RoboDK station: Kuka Station With Tools and Home.rdk

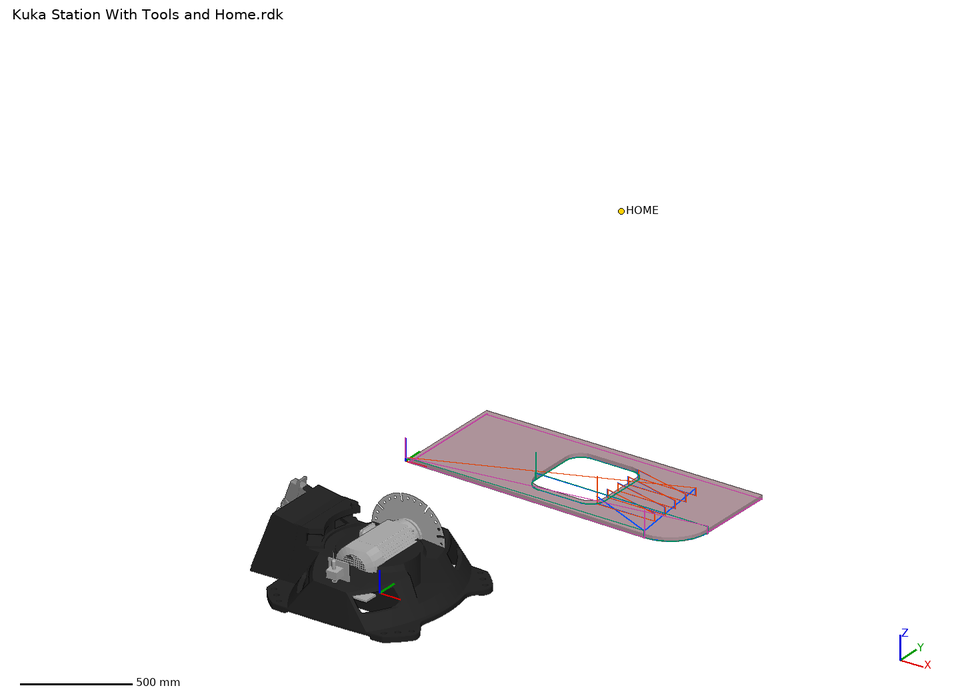
[picture v0: the station drawn from its stored meshes, robots at their saved joint values, targets as dots, program paths as lines]
Station Kuka Station With Tools and Home (saved by RoboDK 5.2.1). Poses are relative to the parent item; angles as X-Y-Z fixed-axis rotations.
  - frame KUKA KR 210 R2700 extra Base at (0, 0, 0) mm
    - robot KUKA KR 210 R2700 extra: 6 axes, payload 210 kg, reach 2696 mm, repeatability 0.06 mm, weight 1068 kg
        joint limits [-185, -140, -120, -350, -125, -350] to [185, -5, 155, 350, 125, 350]; home [0, -90, 90, 0, 0, 0]; saved at [-116.395, -62.059, 114.637, 0, 37.421, -295.134]
      - tool Circular Blade Tool, TCP at (0, 220.26, 403) mm, size 400 x 704.6 x 403 mm, geometry from Motor, Nozzle & Router Rig 2000.stl
      - tool Waterjet, TCP at (0, -363, 366) mm, rotated rx 5 ry 0 rz 0 deg
      - tool Router, TCP at (0, 325, 203) mm, rotated rx -90 ry 0 rz 0 deg
  - frame Table 1 at (-700, 1200, -20) mm
    - target HOME (Cartesian target) at (1431, -363, 1784) mm, rotated rx 0 ry 90 rz -5 deg; joints [0, -90, 90, 0, 0, 0] of KUKA KR 210 R2700 extra
  - object Top1500 US 380Vx400H 5G at (-700, 1200, -40) mm, size 1500 x 625.9 x 20 mm, geometry from Top1500 US 380Vx400H 5G.stl
  - machining project Top1500_US_380Vx400H_5G Settings: C:/Users/Curt Kilian/Dropbox/ROBOT PROGRAMMING TEST FILES/Top1500 US 380Vx400H 5G.dxf | rotZ(0) | rotX(0)*rotY(0) | rotz(0) | onStart | onPathStart | onApproach | onPoint | onRetract | onFinish | SetRPM(%1) | SetTool(%1) | Extruder(%1) | default | default | OutOnMov(%1) | OutOffMov(%1) | onPathFinish | M_RunCode(%1)
  - program Top1500_US_380Vx400H_5G (159 instructions, listed below)
  - machining project Blade Settings: C:/RoboDK/Robot Library/Top1500 US 380Vx400H 5G Blade.ngc | rotZ(0) | rotX(0)*rotY(0) | onStart | onPathStart | onApproach | onPoint | onRetract | onFinish | SetRPM(%1) | SetTool(%1) | Extruder(%1) | default | default | OutOnMov(%1) | OutOffMov(%1) | onPathFinish | M_RunCode(%1)
  - machining project Router Settings: C:/RoboDK/Robot Library/Top1500 US 380Vx400H 5G Router.ngc | rotZ(0) | rotX(0)*rotY(0) | rotz(0) | onStart | onPathStart | onApproach | onPoint | onRetract | onFinish | SetRPM(%1) | SetTool(%1) | Extruder(%1) | default | default | OutOnMov(%1) | OutOffMov(%1) | onPathFinish | M_RunCode(%1)
  - machining project Waterjet Settings: C:/RoboDK/Robot Library/Top1500 US 380Vx400H 5G Waterjet.ngc | rotZ(0) | rotX(0)*rotY(0) | rotz(0) | onStart | onPathStart | onApproach | onPoint | onRetract | onFinish | SetRPM(%1) | SetTool(%1) | Extruder(%1) | default | default | OutOnMov(%1) | OutOffMov(%1) | onPathFinish | M_RunCode(%1)
  - program Router (67 instructions, listed below)
  - program Waterjet (58 instructions, listed below)
  - program Blade (58 instructions, listed below)
  - program Prog2 (3 instructions, listed below)
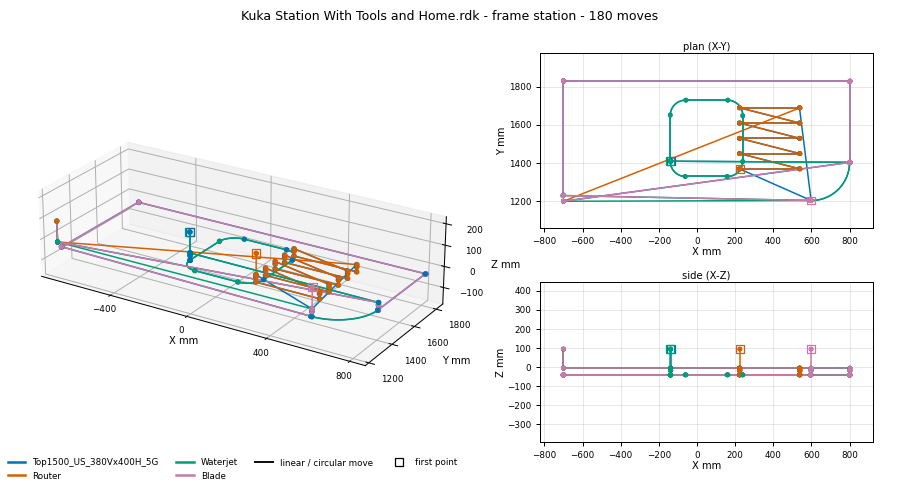
[picture p0: tool path of Kuka Station With Tools and Home.rdk in frame station, 180 of 180 moves have a stored position in this frame; points joined in program order, loops and branches not executed]

--- program Top1500_US_380Vx400H_5G (robot KUKA KR 210 R2700 extra) ---
  Smooth(1)
  Set speed (1000.0 mm/s)
  Set Ref.: Table 1
  Set Tool: Circular Blade Tool
  Show Circular Blade Tool
  MoveJ 1 to (562.5, 210, 115) mm, rotated rx 180 ry 0 rz -67.5 deg; joints [-87.471, -64.949, 119.715, 0, 35.234, 25.029]
  MoveL 2 to (562.5, 210, 115) mm, rotated rx 180 ry 0 rz -67.5 deg; joints [-87.471, -64.949, 119.715, 0, 35.234, 25.029]
  MoveL 3 to (562.5, 210, 15) mm, rotated rx 180 ry 0 rz -67.5 deg; joints [-87.471, -59.92, 119.657, 0, 30.263, 25.029]
  MoveL 4 to (562.5, 210, 15) mm, rotated rx 180 ry 0 rz -67.5 deg; joints [-87.471, -59.92, 119.657, 0, 30.263, 25.029]
  Call SetTool(1)
  Call M_RunCode(6)
  Call SetRPM(6000.0)
  Set speed (1000.0 mm/s)
  MoveL 5 to (562.5, 210, 15) mm, rotated rx 180 ry 0 rz -67.5 deg; joints [-87.471, -59.92, 119.657, 0, 30.263, 25.029]
  Call M_RunCode(3)
  MoveL 6 to (562.5, 210, 3) mm, rotated rx 180 ry 0 rz -67.5 deg; joints [-87.471, -59.3, 119.617, 0, 29.683, 25.029]
  Set speed (2.5 mm/s)
  MoveL 7 to (562.5, 210, -21) mm, rotated rx 180 ry 0 rz -90 deg; joints [-86.641, -60.19, 124.11, 0, 26.081, 3.359]
  Set speed (6.7 mm/s)
  MoveC 8 to (561.77, 211.77, -21) mm, rotated rx 180 ry 0 rz -45 deg; joints [-89.36, -56.144, 115.469, 0, 30.675, 45.64] to (560, 212.5, -21) mm, rotated rx -180 ry 0 rz 0 deg; joints [-94.901, -54.195, 111.374, 0, 32.821, 85.099]
  Set speed (2.5 mm/s)
  MoveL 9 to (560, 212.5, -20) mm, rotated rx 180 ry 0 rz 0 deg; joints [-94.901, -54.241, 111.378, 0, 32.863, 85.099]
  Set speed (6.7 mm/s)
  MoveL 10 to (560, 452.5, -20) mm, rotated rx 180 ry 0 rz -1.79 deg; joints [-94.066, -47.201, 96.831, 0, 40.37, 84.144]
  MoveC 11 to (574.27, 495.67, -20) mm, rotated rx 180 ry 0 rz -100.79 deg; joints [-86.864, -53.733, 110.317, 0, 33.416, -7.654] to (642.5, 530, -20) mm, rotated rx -180 ry 0 rz 178.21 deg; joints [-92.442, -57.698, 118.657, 0, 29.041, -94.232]
  MoveL 12 to (862.5, 530, -20) mm, rotated rx 180 ry 0 rz 178.21 deg; joints [-84.115, -57.523, 118.285, 0, 29.238, -85.905]
  MoveC 13 to (918.34, 504.8, -20) mm, rotated rx -180 ry 0 rz 133.21 deg; joints [-87.87, -56.531, 116.186, 0, 30.345, -134.66] to (940, 447.5, -20) mm, rotated rx -180 ry 0 rz 88.21 deg; joints [-89.313, -53.801, 110.459, 0, 33.342, -181.103]
  MoveL 14 to (940, 207.5, -20) mm, rotated rx -180 ry 0 rz 88.21 deg; joints [-89.196, -60.194, 124.001, 0, 26.193, -180.986]
  MoveC 15 to (914.8, 151.66, -20) mm, rotated rx -180 ry 0 rz 43.21 deg; joints [-87.577, -57.636, 118.526, 0, 29.11, -224.367] to (857.5, 130, -20) mm, rotated rx -180 ry 0 rz -1.79 deg; joints [-83.947, -56.43, 115.972, 0, 30.458, -265.737]
  MoveL 16 to (637.5, 130, -20) mm, rotated rx -180 ry 0 rz -1.79 deg; joints [-92.055, -56.636, 116.408, 0, 30.228, -273.845]
  MoveC 17 to (581.66, 155.2, -20) mm, rotated rx -180 ry 0 rz -26.79 deg; joints [-90.704, -56.615, 116.364, 0, 30.251, -297.494] to (560, 212.5, -20) mm, rotated rx 180 ry 0 rz -71.79 deg; joints [-87.324, -58.439, 120.233, 0, 28.205, -339.114]
  MoveC 18 to (561.2, 212.2, -20) mm, rotated rx -180 ry 0 rz 34.08 deg; joints [-99.338, -54.871, 112.695, 0, 32.176, -245.261] to (562.5, 210, -20) mm, rotated rx -180 ry 0 rz 50 deg; joints [-101.165, -55.817, 114.681, 0, 31.136, -231.165]
  Set speed (2.5 mm/s)
  MoveL 19 to (562.5, 210, 3) mm, rotated rx -180 ry 0 rz 90 deg; joints [-104.237, -60.41, 121.896, 0, 28.514, -194.237]
  Set speed (1000.0 mm/s)
  MoveL 20 to (562.5, 210, 15) mm, rotated rx -180 ry 0 rz 90 deg; joints [-104.237, -61.052, 121.937, 0, 29.115, -194.237]
  Call M_RunCode(9)
  MoveL 21 to (1502.5, 204.04, 15) mm, rotated rx -180 ry 0 rz 90 deg; joints [-67.477, -59.245, 118.299, 0, 30.946, -157.477]
  Call M_RunCode(3)
  MoveL 22 to (1502.5, 204.04, 3) mm, rotated rx -180 ry 0 rz 90 deg; joints [-67.477, -58.638, 118.26, 0, 30.378, -157.477]
  Set speed (2.5 mm/s)
  MoveL 23 to (1502.5, 204.04, -21) mm, rotated rx -180 ry 0 rz 90 deg; joints [-67.477, -57.415, 118.161, 0, 29.254, -157.477]
  Set speed (6.7 mm/s)
  MoveC 24 to (1501.77, 202.27, -21) mm, rotated rx -180 ry 0 rz 45 deg; joints [-67.479, -52.847, 108.561, 0, 34.286, -202.479] to (1500, 201.54, -21) mm, rotated rx -180 ry 0 rz 0 deg; joints [-63.744, -49.282, 101.181, 0, 38.1, -243.744]
  Set speed (2.5 mm/s)
  MoveL 25 to (1500, 201.54, -20) mm, rotated rx -180 ry 0 rz 0 deg; joints [-63.744, -49.323, 101.185, 0, 38.138, -243.744]
  Set speed (6.7 mm/s)
  MoveC 26 to (1438.21, 59.46, -20) mm, rotated rx 180 ry 0 rz -45.57 deg; joints [-57.647, -53.268, 109.347, 0, 33.921, -283.22] to (1293.5, 4.13, -20) mm, rotated rx 180 ry 0 rz -91.15 deg; joints [-55.853, -59.299, 122.075, 0, 27.224, -326.999]
  MoveC 27 to (1295.17, 6.46, -20) mm, rotated rx -180 ry 0 rz 34.3 deg; joints [-71.26, -58.874, 121.165, 0, 27.71, -216.958] to (1298.5, 4.08, -20) mm, rotated rx -180 ry 0 rz -19.86 deg; joints [-64.494, -56.3, 115.7, 0, 30.601, -264.351]
  Set speed (2.5 mm/s)
  MoveL 28 to (1298.5, 4.08, 3) mm, rotated rx 180 ry 0 rz 0.14 deg; joints [-67.227, -57.955, 116.863, 0, 31.092, -247.084]
  Set speed (1000.0 mm/s)
  MoveL 29 to (1298.5, 4.08, 15) mm, rotated rx -180 ry 0 rz 0.14 deg; joints [-67.227, -58.55, 116.902, 0, 31.648, -247.084]
  Call M_RunCode(9)
  MoveL 30 to (922.59, 170, 15) mm, rotated rx 180 ry 0 rz 0.14 deg; joints [-82.052, -56.815, 113.421, 0, 33.394, -261.908]
  Call M_RunCode(3)
  MoveL 31 to (922.59, 170, 3) mm, rotated rx -180 ry 0 rz 0.14 deg; joints [-82.052, -56.249, 113.384, 0, 32.866, -261.908]
  Set speed (2.5 mm/s)
  MoveL 32 to (922.59, 170, -20) mm, rotated rx -180 ry 0 rz 0.14 deg; joints [-82.052, -55.156, 113.293, 0, 31.863, -261.908]
  Set speed (6.7 mm/s)
  MoveL 33 to (1237.5, 170, -20) mm, rotated rx 180 ry 0 rz 0.14 deg; joints [-71.343, -53.125, 109.049, 0, 34.075, -251.2]
  Set speed (2.5 mm/s)
  MoveL 34 to (1237.5, 170, 3) mm, rotated rx -180 ry 0 rz 0.14 deg; joints [-71.343, -54.159, 109.137, 0, 35.022, -251.2]
  Set speed (1000.0 mm/s)
  MoveL 35 to (1237.5, 170, 15) mm, rotated rx -180 ry 0 rz 0.14 deg; joints [-71.343, -54.695, 109.173, 0, 35.522, -251.2]
  Call M_RunCode(9)
  MoveL 36 to (922.59, 250, 15) mm, rotated rx 180 ry 0 rz 0.14 deg; joints [-82.428, -54.503, 108.789, 0, 35.714, -262.285]
  Call M_RunCode(3)
  MoveL 37 to (922.59, 250, 3) mm, rotated rx 180 ry 0 rz 0.14 deg; joints [-82.428, -53.97, 108.753, 0, 35.217, -262.285]
  Set speed (2.5 mm/s)
  MoveL 38 to (922.59, 250, -20) mm, rotated rx -180 ry 0 rz 0.14 deg; joints [-82.428, -52.94, 108.666, 0, 34.274, -262.285]
  Set speed (6.7 mm/s)
  MoveL 39 to (1237.5, 250, -20) mm, rotated rx -180 ry 0 rz 0.14 deg; joints [-72.179, -50.93, 104.499, 0, 36.431, -252.035]
  Set speed (2.5 mm/s)
  MoveL 40 to (1237.5, 250, 3) mm, rotated rx -180 ry 0 rz 0.14 deg; joints [-72.179, -51.91, 104.584, 0, 37.326, -252.035]
  Set speed (1000.0 mm/s)
  MoveL 41 to (1237.5, 250, 15) mm, rotated rx -180 ry 0 rz 0.14 deg; joints [-72.179, -52.417, 104.62, 0, 37.798, -252.035]
  Call M_RunCode(9)
  MoveL 42 to (922.59, 330, 15) mm, rotated rx -180 ry 0 rz 0.14 deg; joints [-82.77, -52.117, 104.02, 0, 38.097, -262.627]
  Call M_RunCode(3)
  MoveL 43 to (922.59, 330, 3) mm, rotated rx -180 ry 0 rz 0.14 deg; joints [-82.77, -51.613, 103.985, 0, 37.629, -262.627]
  Set speed (2.5 mm/s)
  MoveL 44 to (922.59, 330, -20) mm, rotated rx 180 ry 0 rz 0.14 deg; joints [-82.77, -50.64, 103.9, 0, 36.74, -262.627]
  Set speed (6.7 mm/s)
  MoveL 45 to (1237.5, 330, -20) mm, rotated rx -180 ry 0 rz 0.14 deg; joints [-72.945, -48.643, 99.787, 0, 38.856, -252.802]
  Set speed (2.5 mm/s)
  MoveL 46 to (1237.5, 330, 3) mm, rotated rx -180 ry 0 rz 0.14 deg; joints [-72.945, -49.574, 99.87, 0, 39.703, -252.802]
  Set speed (1000.0 mm/s)
  MoveL 47 to (1237.5, 330, 15) mm, rotated rx -180 ry 0 rz 0.14 deg; joints [-72.945, -50.055, 99.905, 0, 40.15, -252.802]
  Call M_RunCode(9)
  MoveL 48 to (922.59, 410, 15) mm, rotated rx -180 ry 0 rz 0.14 deg; joints [-83.083, -49.648, 99.092, 0, 40.555, -262.94]
  Call M_RunCode(3)
  MoveL 49 to (922.59, 410, 3) mm, rotated rx -180 ry 0 rz 0.14 deg; joints [-83.083, -49.17, 99.058, 0, 40.112, -262.94]
  Set speed (2.5 mm/s)
  MoveL 50 to (922.59, 410, -20) mm, rotated rx -180 ry 0 rz 0.14 deg; joints [-83.083, -48.247, 98.975, 0, 39.272, -262.94]
  Set speed (6.7 mm/s)
  MoveL 51 to (1237.5, 410, -20) mm, rotated rx -180 ry 0 rz 0.14 deg; joints [-73.65, -46.253, 94.891, 0, 41.362, -253.506]
  Set speed (2.5 mm/s)
  MoveL 52 to (1237.5, 410, 3) mm, rotated rx 180 ry 0 rz 0.14 deg; joints [-73.65, -47.14, 94.973, 0, 42.166, -253.506]
  Set speed (1000.0 mm/s)
  MoveL 53 to (1237.5, 410, 15) mm, rotated rx -180 ry 0 rz 0.14 deg; joints [-73.65, -47.598, 95.008, 0, 42.591, -253.506]
  Call M_RunCode(9)
  MoveL 54 to (922.59, 490, 15) mm, rotated rx -180 ry 0 rz 0.14 deg; joints [-83.37, -47.082, 93.98, 0, 43.102, -263.227]
  Call M_RunCode(3)
  MoveL 55 to (922.59, 490, 3) mm, rotated rx 180 ry 0 rz 0.14 deg; joints [-83.37, -46.628, 93.946, 0, 42.682, -263.227]
  Set speed (2.5 mm/s)
  MoveL 56 to (922.59, 490, -20) mm, rotated rx -180 ry 0 rz 0.14 deg; joints [-83.37, -45.75, 93.864, 0, 41.886, -263.227]
  Set speed (6.7 mm/s)
  MoveL 57 to (1237.5, 490, -20) mm, rotated rx 180 ry 0 rz 0.14 deg; joints [-74.3, -43.747, 89.783, 0, 43.964, -254.157]
  Set speed (2.5 mm/s)
  MoveL 58 to (1237.5, 490, 3) mm, rotated rx -180 ry 0 rz 0.14 deg; joints [-74.3, -44.594, 89.865, 0, 44.729, -254.157]
  Set speed (1000.0 mm/s)
  MoveL 59 to (1237.5, 490, 15) mm, rotated rx -180 ry 0 rz 0.14 deg; joints [-74.3, -45.032, 89.899, 0, 45.133, -254.157]
  Call M_RunCode(9)
  MoveL 60 to (1298.5, 4.08, 15) mm, rotated rx 180 ry 0 rz 0.14 deg; joints [-67.227, -58.55, 116.902, 0, 31.648, -247.084]
  Call M_RunCode(3)
  MoveL 61 to (1298.5, 4.08, 3) mm, rotated rx 180 ry 0 rz 0.14 deg; joints [-67.227, -57.955, 116.863, 0, 31.092, -247.084]
  Set speed (2.5 mm/s)
  MoveL 62 to (1298.5, 4.08, -21) mm, rotated rx -180 ry 0 rz 0.14 deg; joints [-67.227, -56.757, 116.765, 0, 29.992, -247.084]
  Set speed (6.7 mm/s)
  MoveC 63 to (1296.03, 6.61, -21) mm, rotated rx -180 ry 0 rz 90.14 deg; joints [-72.695, -63.82, 132.107, 0, 21.713, -162.551] to (1293.5, 4.13, -21) mm, rotated rx -180 ry 0 rz -179.86 deg; joints [-58.877, -66.405, 138.049, 0, 18.356, -58.734]
  Set speed (2.5 mm/s)
  MoveL 64 to (1293.5, 4.13, -20) mm, rotated rx 180 ry 0 rz -179.86 deg; joints [-58.877, -66.479, 138.055, 0, 18.424, -58.734]
  Set speed (6.7 mm/s)
  MoveL 65 to (-2.5, 30.05, -20) mm, rotated rx -180 ry 0 rz -179.86 deg; joints [-124.805, -64.664, 133.87, 0, 20.794, -124.662]
  Set speed (2.5 mm/s)
  MoveL 66 to (-2.5, 30.05, -21) mm, rotated rx -180 ry 0 rz -179.86 deg; joints [-124.805, -64.597, 133.864, 0, 20.733, -124.662]
  Set speed (6.7 mm/s)
  MoveC 67 to (-1.75, 31.79, -21) mm, rotated rx -180 ry 0 rz 135.7 deg; joints [-128.538, -61.169, 126.236, 0, 24.933, -172.838] to (0, 32.5, -21) mm, rotated rx -180 ry 0 rz 91.26 deg; joints [-126.854, -57.037, 117.359, 0, 29.679, -215.593]
  Set speed (2.5 mm/s)
  MoveL 68 to (0, 32.5, -20) mm, rotated rx -180 ry 0 rz 91.26 deg; joints [-126.854, -57.088, 117.363, 0, 29.725, -215.593]
  Set speed (6.7 mm/s)
  MoveL 69 to (0, 632.5, -20) mm, rotated rx -180 ry 0 rz 91.26 deg; joints [-116.725, -41.638, 85.502, 0, 46.137, -205.464]
  Set speed (2.5 mm/s)
  MoveL 70 to (0, 632.5, -21) mm, rotated rx -180 ry 0 rz 91.26 deg; joints [-116.725, -41.603, 85.498, 0, 46.105, -205.464]
  Set speed (6.7 mm/s)
  MoveC 71 to (1.77, 631.77, -21) mm, rotated rx -180 ry 0 rz 46.26 deg; joints [-113.371, -37.427, 77.053, 0, 50.374, -247.11] to (2.5, 630, -21) mm, rotated rx -180 ry 0 rz 1.26 deg; joints [-108.91, -37.206, 76.607, 0, 50.598, -287.649]
  Set speed (2.5 mm/s)
  MoveL 72 to (2.5, 630, -20) mm, rotated rx 180 ry 0 rz 1.26 deg; joints [-108.91, -37.239, 76.612, 0, 50.628, -287.649]
  Set speed (6.7 mm/s)
  MoveL 73 to (1502.5, 630, -20) mm, rotated rx -180 ry 0 rz 1.26 deg; joints [-68.741, -35.972, 74.058, 0, 51.913, -247.48]
  Set speed (2.5 mm/s)
  MoveL 74 to (1502.5, 630, -21) mm, rotated rx -180 ry 0 rz 1.26 deg; joints [-68.741, -35.939, 74.054, 0, 51.885, -247.48]
  Set speed (6.7 mm/s)
  MoveC 75 to (1501.77, 628.23, -21) mm, rotated rx 180 ry 0 rz -43.74 deg; joints [-64.356, -35.758, 73.69, 0, 52.068, -288.095] to (1500, 627.5, -21) mm, rotated rx 180 ry 0 rz -88.74 deg; joints [-60.892, -39.799, 81.844, 0, 47.955, -329.631]
  Set speed (2.5 mm/s)
  MoveL 76 to (1500, 627.5, -20) mm, rotated rx 180 ry 0 rz -88.74 deg; joints [-60.892, -39.834, 81.849, 0, 47.985, -329.631]
  Set speed (6.7 mm/s)
  MoveL 77 to (1500, 201.54, -20) mm, rotated rx 180 ry 0 rz -88.74 deg; joints [-54.043, -51.428, 105.528, 0, 35.9, -322.782]
  MoveC 78 to (1501.77, 202.27, -20) mm, rotated rx 180 ry 0 rz -43.74 deg; joints [-58.574, -48.672, 99.847, 0, 38.825, -282.313] to (1502.5, 204.04, -20) mm, rotated rx -180 ry 0 rz 1.26 deg; joints [-63.845, -49.288, 101.113, 0, 38.175, -242.584]
  Set speed (2.5 mm/s)
  MoveL 79 to (1502.5, 204.04, 3) mm, rotated rx 180 ry 0 rz 1.26 deg; joints [-63.845, -50.232, 101.197, 0, 39.035, -242.584]
  Set speed (1000.0 mm/s)
  MoveL 80 to (1502.5, 204.04, 15) mm, rotated rx -180 ry 0 rz 1.26 deg; joints [-63.845, -50.72, 101.232, 0, 39.489, -242.584]
  Call M_RunCode(9)
  MoveL 81 to (0, 0, 15) mm, rotated rx 180 ry 0 rz 1.26 deg; joints [-116.395, -57.394, 114.582, 0, 32.812, -295.134]
  MoveL 82 to (0, 0, 15) mm, rotated rx 180 ry 0 rz 1.26 deg; joints [-116.395, -57.394, 114.582, 0, 32.812, -295.134]
  MoveL 83 to (0, 0, 115) mm, rotated rx 180 ry 0 rz 1.26 deg; joints [-116.395, -62.059, 114.637, 0, 37.421, -295.134]
  Call M_RunCode(2)

--- program Router (robot KUKA KR 210 R2700 extra) ---
  Smooth(1)
  Set speed (1000.0 mm/s)
  Set Ref.: Table 1
  Set Tool: Router
  Show Router
  MoveJ 1 to (925.09, 170, 115) mm, rotated rx -180 ry 0 rz -180 deg; joints [-82.825, -42.749, 100.39, 8.476, 122.075, -85.475]
  MoveL 2 to (925.09, 170, 115) mm, rotated rx -180 ry 0 rz -180 deg; joints [-82.825, -42.749, 100.39, 8.476, 122.075, -85.475]
  MoveL 3 to (925.09, 170, 15) mm, rotated rx -180 ry 0 rz -180 deg; joints [-82.825, -38.29, 99.098, 8.206, 118.942, -86.008]
  MoveL 4 to (925.09, 170, 15) mm, rotated rx -180 ry 0 rz -180 deg; joints [-82.825, -38.29, 99.098, 8.206, 118.942, -86.008]
  Call SetTool(10)
  Call M_RunCode(6)
  Call SetRPM(6000.0)
  Set speed (1000.0 mm/s)
  MoveL 5 to (925.09, 170, 15) mm, rotated rx -180 ry 0 rz -180 deg; joints [-82.825, -38.29, 99.098, 8.206, 118.942, -86.008]
  Call M_RunCode(3)
  MoveL 6 to (925.09, 170, 3) mm, rotated rx -180 ry 0 rz -180 deg; joints [-82.825, -37.747, 98.915, 8.178, 118.586, -86.067]
  Set speed (2.5 mm/s)
  MoveL 7 to (925.09, 170, -20) mm, rotated rx -180 ry 0 rz -180 deg; joints [-82.825, -36.704, 98.547, 8.126, 117.917, -86.175]
  MoveL 8 to (1240, 170, -20) mm, rotated rx 180 ry 0 rz 180 deg; joints [-73.195, -35.178, 94.456, 19.357, 119.278, -80.251]
  MoveL 9 to (1240, 170, 3) mm, rotated rx -180 ry 0 rz 180 deg; joints [-73.195, -36.186, 94.82, 19.479, 119.886, -80.005]
  Set speed (1000.0 mm/s)
  MoveL 10 to (1240, 170, 15) mm, rotated rx -180 ry 0 rz -14.25 deg; joints [-65.63, -47.18, 138.68, 190.12, 91.477, -89.736]
  Call M_RunCode(9)
  MoveL 11 to (925.09, 250, 15) mm, rotated rx -180 ry 0 rz -14.25 deg; joints [-83.331, -47.144, 139.017, 172.411, 91.857, -90.247]
  Call M_RunCode(3)
  MoveL 12 to (925.09, 250, 3) mm, rotated rx 180 ry 0 rz -14.25 deg; joints [-83.331, -46.199, 138.732, 172.408, 92.511, -90.335]
  Set speed (2.5 mm/s)
  MoveL 13 to (925.09, 250, -20) mm, rotated rx -180 ry 0 rz 180 deg; joints [-83.129, -34.844, 93.582, 8.024, 121.012, -85.846]
  MoveL 14 to (1240, 250, -20) mm, rotated rx 180 ry 0 rz 180 deg; joints [-73.877, -33.246, 89.489, 19.173, 122.263, -79.485]
  MoveL 15 to (1240, 250, 3) mm, rotated rx -180 ry 0 rz 180 deg; joints [-73.877, -34.217, 89.851, 19.301, 122.839, -79.247]
  Set speed (1000.0 mm/s)
  MoveL 16 to (1240, 250, 15) mm, rotated rx -180 ry 0 rz -14.25 deg; joints [-67.3, -47.34, 135.225, 188.452, 87.908, -90.311]
  Call M_RunCode(9)
  MoveL 17 to (925.09, 330, 15) mm, rotated rx 180 ry 0 rz -14.25 deg; joints [-83.802, -47.34, 135.279, 171.939, 87.959, -89.711]
  Call M_RunCode(3)
  MoveL 18 to (925.09, 330, 3) mm, rotated rx 180 ry 0 rz -14.25 deg; joints [-83.802, -46.462, 135.015, 171.942, 88.567, -89.797]
  Set speed (2.5 mm/s)
  MoveL 19 to (925.09, 330, -20) mm, rotated rx -180 ry 0 rz 180 deg; joints [-83.409, -32.809, 88.393, 7.973, 124.157, -85.503]
  MoveL 20 to (1240, 330, -20) mm, rotated rx -180 ry 0 rz -160 deg; joints [-78.333, -32.745, 88.233, 36.817, 118.831, -70.152]
  MoveL 21 to (1240, 330, 3) mm, rotated rx 180 ry 0 rz -160 deg; joints [-78.333, -33.708, 88.595, 37.018, 119.311, -69.739]
  Set speed (1000.0 mm/s)
  MoveL 22 to (1240, 330, 15) mm, rotated rx 180 ry 0 rz -14.25 deg; joints [-68.766, -47.168, 131.631, 187.013, 84.504, -90.675]
  Call M_RunCode(9)
  MoveL 23 to (925.09, 410, 15) mm, rotated rx -180 ry 0 rz -14.25 deg; joints [-84.21, -47.15, 131.423, 171.494, 84.336, -89.154]
  Call M_RunCode(3)
  MoveL 24 to (925.09, 410, 3) mm, rotated rx 180 ry 0 rz -14.25 deg; joints [-84.21, -46.33, 131.176, 171.502, 84.902, -89.239]
  Set speed (2.5 mm/s)
  MoveL 25 to (925.09, 410, -20) mm, rotated rx -180 ry 0 rz -160 deg; joints [-87.652, -31.618, 85.445, 26.989, 123.086, -74.463]
  MoveL 26 to (1240, 410, -20) mm, rotated rx 180 ry 0 rz -160 deg; joints [-78.787, -30.55, 82.849, 37.446, 121.535, -68.172]
  MoveL 27 to (1240, 410, 3) mm, rotated rx -180 ry 0 rz -160 deg; joints [-78.787, -31.48, 83.212, 37.66, 121.985, -67.765]
  Set speed (1000.0 mm/s)
  MoveL 28 to (1240, 410, 15) mm, rotated rx 180 ry 0 rz -14.25 deg; joints [-70.061, -46.714, 127.907, 185.752, 81.237, -90.879]
  Call M_RunCode(9)
  MoveL 29 to (925.09, 490, 15) mm, rotated rx 180 ry 0 rz -14.25 deg; joints [-84.569, -46.643, 127.455, 171.065, 80.922, -88.579]
  Call M_RunCode(3)
  MoveL 30 to (925.09, 490, 3) mm, rotated rx -180 ry 0 rz -14.25 deg; joints [-84.569, -45.876, 127.222, 171.078, 81.45, -88.663]
  Set speed (2.5 mm/s)
  MoveL 31 to (925.09, 490, -20) mm, rotated rx -180 ry 0 rz 140 deg; joints [-76.2, -29.713, 80.842, 327.707, 124.27, -109.589]
  MoveL 32 to (1240, 490, -20) mm, rotated rx -180 ry 0 rz 120 deg; joints [-64.593, -28.718, 78.484, 317.905, 122.122, -115.658]
  MoveL 33 to (1240, 490, 3) mm, rotated rx 180 ry 0 rz 120 deg; joints [-64.593, -29.627, 78.851, 317.675, 122.523, -116.089]
  Set speed (1000.0 mm/s)
  MoveL 34 to (1240, 490, 15) mm, rotated rx 180 ry 0 rz 21.56 deg; joints [-61.941, -44.525, 117.868, 230.829, 79.299, -102.839]
  Call M_RunCode(9)
  MoveL 35 to (0, 0, 15) mm, rotated rx -180 ry 0 rz 21.56 deg; joints [-123.96, -46.528, 142.379, 167.539, 95.714, -91.26]
  MoveL 36 to (0, 0, 15) mm, rotated rx -180 ry 0 rz 21.56 deg; joints [-123.96, -46.528, 142.379, 167.539, 95.714, -91.26]
  MoveL 37 to (0, 0, 115) mm, rotated rx 180 ry 0 rz 21.56 deg; joints [-123.96, -55.295, 144.61, 167.601, 89.332, -89.853]
  Call M_RunCode(2)

--- program Waterjet (robot KUKA KR 210 R2700 extra) ---
  Smooth(1)
  Set speed (1000.0 mm/s)
  Set Ref.: Table 1
  Set Tool: Waterjet
  Show Waterjet
  MoveJ 1 to (560.5, 210, 115) mm, rotated rx 180 ry 0 rz -180 deg; joints [-94.634, -57.138, 106.366, 0.69, 35.79, -95.176]
  MoveL 2 to (560.5, 210, 115) mm, rotated rx 180 ry 0 rz -180 deg; joints [-94.634, -57.138, 106.366, 0.69, 35.79, -95.176]
  MoveL 3 to (560.5, 210, 15) mm, rotated rx -180 ry 0 rz -180 deg; joints [-94.634, -52.933, 106.28, 0.768, 31.671, -95.271]
  MoveL 4 to (560.5, 210, 15) mm, rotated rx -180 ry 0 rz -180 deg; joints [-94.634, -52.933, 106.28, 0.768, 31.671, -95.271]
  Call SetTool(2)
  Call M_RunCode(6)
  Call SetRPM(6000.0)
  Set speed (1000.0 mm/s)
  MoveL 5 to (560.5, 210, 15) mm, rotated rx -180 ry 0 rz -180 deg; joints [-94.634, -52.933, 106.28, 0.768, 31.671, -95.271]
  Call M_RunCode(3)
  MoveL 6 to (560.5, 210, 3) mm, rotated rx -180 ry 0 rz -180 deg; joints [-94.634, -52.414, 106.241, 0.779, 31.192, -95.283]
  Set speed (2.5 mm/s)
  MoveL 7 to (560.5, 210, -21) mm, rotated rx 180 ry 0 rz -180 deg; joints [-94.634, -51.368, 106.142, 0.801, 30.244, -95.309]
  Set speed (4.2 mm/s)
  MoveC 8 to (560.35, 210.35, -21) mm, rotated rx -180 ry 0 rz 180 deg; joints [-94.638, -51.357, 106.121, 0.801, 30.255, -95.313] to (560, 210.5, -21) mm, rotated rx -180 ry 0 rz -180 deg; joints [-94.649, -51.352, 106.11, 0.803, 30.261, -95.326]
  Set speed (2.5 mm/s)
  MoveL 9 to (560, 210.5, -20) mm, rotated rx -180 ry 0 rz -180 deg; joints [-94.649, -51.396, 106.115, 0.802, 30.3, -95.324]
  Set speed (4.2 mm/s)
  MoveL 10 to (560, 450.5, -20) mm, rotated rx 180 ry 0 rz 180 deg; joints [-94.083, -44.054, 90.955, 0.576, 38.114, -94.52]
  MoveC 11 to (583.79, 506.92, -20) mm, rotated rx 180 ry 0 rz -180 deg; joints [-93.296, -42.224, 87.217, 0.447, 40.016, -93.626] to (640.5, 530, -20) mm, rotated rx 180 ry 0 rz -180 deg; joints [-91.67, -41.519, 85.779, 0.223, 40.742, -91.832]
  MoveL 12 to (860.5, 530, -20) mm, rotated rx 180 ry 0 rz 180 deg; joints [-85.504, -41.331, 85.396, -0.597, 40.951, -85.069]
  MoveC 13 to (916.92, 506.21, -20) mm, rotated rx -180 ry 0 rz -180 deg; joints [-83.862, -41.966, 86.69, -0.825, 40.307, -83.256] to (940, 449.5, -20) mm, rotated rx 180 ry 0 rz -180 deg; joints [-83.021, -43.77, 90.372, -0.976, 38.438, -82.282]
  MoveL 14 to (940, 209.5, -20) mm, rotated rx -180 ry 0 rz -180 deg; joints [-82.059, -51.108, 105.514, -1.353, 30.649, -80.924]
  MoveC 15 to (916.21, 153.08, -20) mm, rotated rx 180 ry 0 rz -180 deg; joints [-82.597, -52.794, 109.04, -1.336, 28.801, -81.454] to (859.5, 130, -20) mm, rotated rx -180 ry 0 rz -180 deg; joints [-84.448, -53.613, 110.763, -1.033, 27.877, -83.556]
  MoveL 16 to (639.5, 130, -20) mm, rotated rx -180 ry 0 rz 180 deg; joints [-92.111, -53.796, 111.149, 0.396, 27.651, -92.455]
  MoveC 17 to (583.08, 153.79, -20) mm, rotated rx 180 ry 0 rz -180 deg; joints [-94.017, -53.051, 109.581, 0.734, 28.484, -94.647] to (560, 210.5, -20) mm, rotated rx -180 ry 0 rz -180 deg; joints [-94.649, -51.396, 106.115, 0.802, 30.3, -95.324]
  MoveC 18 to (560.35, 210.35, -20) mm, rotated rx 180 ry 0 rz -180 deg; joints [-94.638, -51.401, 106.125, 0.8, 30.295, -95.312] to (560.5, 210, -20) mm, rotated rx 180 ry 0 rz -180 deg; joints [-94.634, -51.412, 106.147, 0.8, 30.283, -95.308]
  Set speed (2.5 mm/s)
  MoveL 19 to (560.5, 210, 3) mm, rotated rx -180 ry 0 rz -180 deg; joints [-94.634, -52.414, 106.241, 0.779, 31.192, -95.283]
  Set speed (1000.0 mm/s)
  MoveL 20 to (560.5, 210, 15) mm, rotated rx -180 ry 0 rz -180 deg; joints [-94.634, -52.933, 106.28, 0.768, 31.671, -95.271]
  Call M_RunCode(9)
  MoveL 21 to (1500.5, 204.04, 15) mm, rotated rx 180 ry 0 rz 180 deg; joints [-64.979, -47.787, 95.944, -3.483, 37.361, -62.293]
  Call M_RunCode(3)
  MoveL 22 to (1500.5, 204.04, 3) mm, rotated rx 180 ry 0 rz 180 deg; joints [-64.979, -47.322, 95.906, -3.517, 36.936, -62.25]
  Set speed (2.5 mm/s)
  MoveL 23 to (1500.5, 204.04, -21) mm, rotated rx 180 ry 0 rz 180 deg; joints [-64.979, -46.385, 95.812, -3.588, 36.094, -62.162]
  Set speed (4.2 mm/s)
  MoveC 24 to (1500.35, 203.69, -21) mm, rotated rx 180 ry 0 rz 180 deg; joints [-64.978, -46.397, 95.836, -3.589, 36.081, -62.16] to (1500, 203.54, -21) mm, rotated rx -180 ry 0 rz -180 deg; joints [-64.986, -46.406, 95.855, -3.589, 36.071, -62.168]
  Set speed (2.5 mm/s)
  MoveL 25 to (1500, 203.54, -20) mm, rotated rx 180 ry 0 rz -180 deg; joints [-64.986, -46.445, 95.859, -3.586, 36.106, -62.172]
  Set speed (4.2 mm/s)
  MoveC 26 to (1439.64, 60.86, -20) mm, rotated rx -180 ry 0 rz -180 deg; joints [-64.8, -51.107, 105.512, -4.116, 31.134, -61.36] to (1295.5, 4.09, -20) mm, rotated rx 180 ry 0 rz 180 deg; joints [-68.543, -54.187, 111.974, -3.944, 27.614, -65.121]
  MoveC 27 to (1296.01, 4.58, -20) mm, rotated rx 180 ry 0 rz -180 deg; joints [-68.532, -54.169, 111.937, -3.943, 27.634, -65.112] to (1296.5, 4.08, -20) mm, rotated rx 180 ry 0 rz -180 deg; joints [-68.51, -54.177, 111.954, -3.948, 27.626, -65.085]
  Set speed (2.5 mm/s)
  MoveL 28 to (1296.5, 4.08, 3) mm, rotated rx 180 ry 0 rz 180 deg; joints [-68.51, -55.255, 112.051, -3.824, 28.604, -65.226]
  Set speed (1000.0 mm/s)
  MoveL 29 to (1296.5, 4.08, 15) mm, rotated rx -180 ry 0 rz 180 deg; joints [-68.51, -55.813, 112.092, -3.762, 29.12, -65.296]
  Call M_RunCode(9)
  MoveL 30 to (0, 0, 15) mm, rotated rx -180 ry 0 rz 180 deg; joints [-114.857, -54.743, 109.93, 4.159, 30.34, -118.365]
  MoveL 31 to (0, 0, 15) mm, rotated rx -180 ry 0 rz 180 deg; joints [-114.857, -54.743, 109.93, 4.159, 30.34, -118.365]
  MoveL 32 to (0, 0, 115) mm, rotated rx -180 ry 0 rz -180 deg; joints [-114.857, -59.143, 110.017, 3.695, 34.642, -117.815]
  Call M_RunCode(2)

--- program Blade (robot KUKA KR 210 R2700 extra) ---
  Smooth(1)
  Set speed (1000.0 mm/s)
  Set Ref.: Table 1
  Set Tool: Circular Blade Tool
  Show Circular Blade Tool
  MoveJ 1 to (1298.5, 4.08, 115) mm, rotated rx 180 ry 0 rz -45.57 deg; joints [-60.906, -63.063, 116.413, 0, 36.65, 73.521]
  MoveL 2 to (1298.5, 4.08, 115) mm, rotated rx 180 ry 0 rz -45.57 deg; joints [-60.906, -63.063, 116.413, 0, 36.65, 73.521]
  MoveL 3 to (1298.5, 4.08, 15) mm, rotated rx 180 ry 0 rz -45.57 deg; joints [-60.906, -58.278, 116.356, 0, 31.922, 73.521]
  MoveL 4 to (1298.5, 4.08, 15) mm, rotated rx 180 ry 0 rz -45.57 deg; joints [-60.906, -58.278, 116.356, 0, 31.922, 73.521]
  Call SetTool(1)
  Call M_RunCode(6)
  Call SetRPM(6000.0)
  Set speed (1000.0 mm/s)
  MoveL 5 to (1298.5, 4.08, 15) mm, rotated rx 180 ry 0 rz -45.57 deg; joints [-60.906, -58.278, 116.356, 0, 31.922, 73.521]
  Call M_RunCode(3)
  MoveL 6 to (1298.5, 4.08, 3) mm, rotated rx -180 ry 0 rz -45.57 deg; joints [-60.906, -57.688, 116.318, 0, 31.371, 73.521]
  Set speed (2.5 mm/s)
  MoveL 7 to (1298.5, 4.08, -21) mm, rotated rx -180 ry 0 rz -0.57 deg; joints [-67.133, -56.729, 116.705, 0, 30.024, 112.294]
  Set speed (6.7 mm/s)
  MoveC 8 to (1296.03, 6.61, -21) mm, rotated rx -180 ry 0 rz 89.43 deg; joints [-72.731, -63.758, 131.968, 0, 21.79, 196.696] to (1293.5, 4.13, -21) mm, rotated rx -180 ry 0 rz 179.43 deg; joints [-58.995, -66.436, 138.122, 0, 18.314, 300.432]
  Set speed (2.5 mm/s)
  MoveL 9 to (1293.5, 4.13, -20) mm, rotated rx 180 ry 0 rz 178.85 deg; joints [-59.09, -66.534, 138.185, 0, 18.349, 299.764]
  Set speed (6.7 mm/s)
  MoveL 10 to (-2.5, 30.05, -20) mm, rotated rx -180 ry 0 rz 178.85 deg; joints [-124.993, -64.598, 133.719, 0, 20.879, 233.861]
  Set speed (2.5 mm/s)
  MoveL 11 to (-2.5, 30.05, -21) mm, rotated rx -180 ry 0 rz 178.86 deg; joints [-124.992, -64.531, 133.715, 0, 20.816, 233.871]
  Set speed (6.7 mm/s)
  MoveC 12 to (-1.75, 31.79, -21) mm, rotated rx -180 ry 0 rz 134.42 deg; joints [-128.561, -61.047, 125.972, 0, 25.076, 185.858] to (0, 32.5, -21) mm, rotated rx -180 ry 0 rz 89.98 deg; joints [-126.746, -56.932, 117.135, 0, 29.797, 143.235]
  Set speed (2.5 mm/s)
  MoveL 13 to (0, 32.5, -20) mm, rotated rx -180 ry 0 rz 90 deg; joints [-126.747, -56.984, 117.143, 0, 29.841, 143.253]
  Set speed (6.7 mm/s)
  MoveL 14 to (0, 632.5, -20) mm, rotated rx -180 ry 0 rz 90 deg; joints [-116.665, -41.487, 85.194, 0, 46.292, 153.335]
  Set speed (2.5 mm/s)
  MoveL 15 to (0, 632.5, -21) mm, rotated rx 180 ry 0 rz 90 deg; joints [-116.665, -41.451, 85.19, 0, 46.261, 153.335]
  Set speed (6.7 mm/s)
  MoveC 16 to (1.77, 631.77, -21) mm, rotated rx -180 ry 0 rz 45 deg; joints [-113.252, -37.357, 76.911, 0, 50.445, 111.748] to (2.5, 630, -21) mm, rotated rx 180 ry 0 rz 0 deg; joints [-108.788, -37.264, 76.724, 0, 50.54, 71.212]
  Set speed (2.5 mm/s)
  MoveL 17 to (2.5, 630, -20) mm, rotated rx 180 ry 0 rz 0 deg; joints [-108.788, -37.297, 76.728, 0, 50.569, 71.212]
  Set speed (6.7 mm/s)
  MoveL 18 to (1502.5, 630, -20) mm, rotated rx 180 ry 0 rz 0 deg; joints [-68.624, -35.9, 73.915, 0, 51.986, 111.376]
  Set speed (2.5 mm/s)
  MoveL 19 to (1502.5, 630, -21) mm, rotated rx 180 ry 0 rz 0 deg; joints [-68.624, -35.867, 73.911, 0, 51.957, 111.376]
  Set speed (6.7 mm/s)
  MoveC 20 to (1501.77, 628.23, -21) mm, rotated rx 180 ry 0 rz -45 deg; joints [-64.237, -35.819, 73.813, 0, 52.006, 70.763] to (1500, 627.5, -21) mm, rotated rx 180 ry 0 rz -90 deg; joints [-60.826, -39.95, 82.151, 0, 47.8, 29.174]
  Set speed (2.5 mm/s)
  MoveL 21 to (1500, 627.5, -20) mm, rotated rx 180 ry 0 rz -90 deg; joints [-60.826, -39.985, 82.155, 0, 47.83, 29.174]
  Set speed (6.7 mm/s)
  MoveL 22 to (1500, 201.54, -20) mm, rotated rx 180 ry 0 rz -90 deg; joints [-53.947, -51.541, 105.763, 0, 35.778, 36.053]
  MoveC 23 to (1501.77, 202.27, -20) mm, rotated rx 180 ry 0 rz -45 deg; joints [-58.426, -48.705, 99.915, 0, 38.79, 76.574] to (1502.5, 204.04, -20) mm, rotated rx -180 ry 0 rz 0 deg; joints [-63.708, -49.222, 100.977, 0, 38.245, 116.292]
  Set speed (2.5 mm/s)
  MoveL 24 to (1502.5, 204.04, 3) mm, rotated rx -180 ry 0 rz 0 deg; joints [-63.708, -50.164, 101.061, 0, 39.104, 116.292]
  Set speed (1000.0 mm/s)
  MoveL 25 to (1502.5, 204.04, 15) mm, rotated rx -180 ry 0 rz 7.73 deg; joints [-64.527, -51.111, 102.011, 0, 39.1, 123.207]
  Call M_RunCode(9)
  MoveL 26 to (0, 0, 15) mm, rotated rx 180 ry 0 rz 7.73 deg; joints [-117.224, -57.124, 114.04, 0, 33.084, 70.509]
  MoveL 27 to (0, 0, 15) mm, rotated rx 180 ry 0 rz 7.73 deg; joints [-117.224, -57.124, 114.04, 0, 33.084, 70.509]
  MoveL 28 to (0, 0, 115) mm, rotated rx -180 ry 0 rz 7.73 deg; joints [-117.224, -61.753, 114.095, 0, 37.658, 70.509]
  Call M_RunCode(2)

--- program Prog2 (robot KUKA KR 210 R2700 extra) ---
  Call Blade
  Call Router
  Call Waterjet
